{attribute addProperty BoxType "EL5001-0000-1016"}
{attribute addProperty Id "Channel_1AT %I*Channel_D09D0F614050WcStateAT %I*WcState_98A4DF7520.250InfoDataAT %I*InfoData_BC63D37F80100"}
{attribute addProperty CRC "325759311"}
{attribute addProperty SizeInBites "122"}
{attribute addProperty SizeInBytes "15.25"}
TYPE EL5001_C393BC80 :
STRUCT
	{attribute addProperty Name "Channel_1"}
	Channel_1 : Channel_D09D0F61;
	{attribute addProperty Name "WcState"}
	WcState : WcState_98A4DF75;
	{attribute addProperty Name "InfoData"}
	InfoData : InfoData_BC63D37F;
END_STRUCT
END_TYPE

(* stored: Version 1.2.0.0, ProductVersion 3.1.4024.9
   DUT EL5001_C393BC80: Id {cd7ca278-5321-4946-8ab9-154816a67fb1} *)
